Staubli VAL3: remSetPPS.pgx

program remSetPPS(string& sArgs[] (dimensions=1), string& sReturn[] (dimensions=1))
begin
  // Set the PPS status in the robot
  //
  logMsg("call remSetPPS")
  call remSetnGlobal(sArgs,nPPS,0,5000,"NOTPPS",sReturn)
end
